TYPE GAIN_SCHEDULED_PID :
STRUCT
	q			:REAL; 	(*gain scheduled parameter for which this PID is optimized*)
	Kp			:REAL;	(*constant for proportional part of the PID*)
	Ki			:REAL;	(*constant for integral part of the PID*)
	Kd			:REAL;	(*constant for derivative part of the PID*)
END_STRUCT
END_TYPE

(* stored: Version 1.1.0.1, ProductVersion 3.1.0.26
   DUT GAIN_SCHEDULED_PID: Id {6ad1baab-7f08-4cb1-b68d-92afca30af89} *)
